Universal Robots PolyScope program: Hospital_small_top.urp

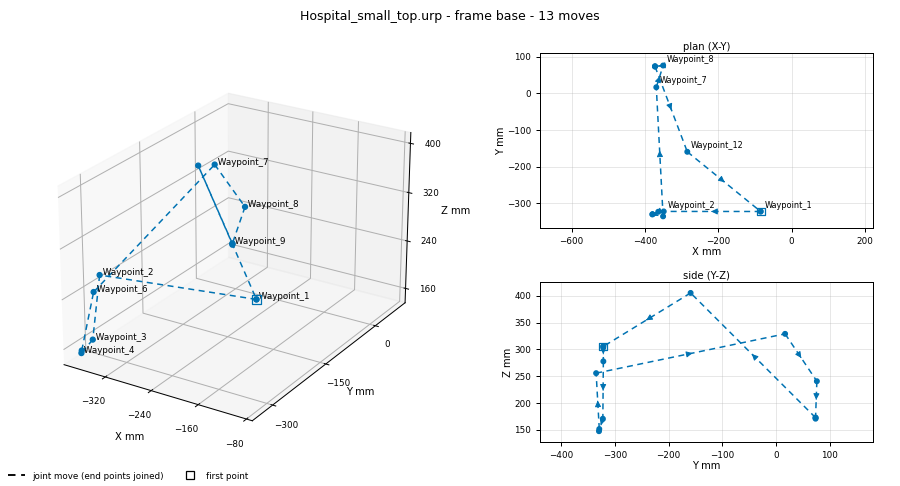
[picture p0: tool path of Hospital_small_top.urp in frame base, 13 of 13 moves have a stored position in this frame; points joined in program order, loops and branches not executed]
Program Hospital_small_top (installation=default directory=/programs/usbdisk/Zahra1 createdIn=5.11.11.1010533 lastSavedIn=5.11.11.1010533 robotSerialNumber=20205300864)
Calibrated DH parameters: a=[-0.000166, -0.243494, -0.153108, 0.000057, -0.000123, 0]; d=[0.151897, -1.34267, 53.988124, -52.514559, 0.085283, 0.092193]; alpha=[1.572472, -0.003756, 0.002824, 1.570807, -1.572621, 0]; deltaTheta=[0, 0.020704, 7.033215, -0.770746, 0.000004, 0]
Robot Program (runOnlyOnce=true)
  MoveJ speed 60 deg/s, acceleration 80 deg/s^2 (useActiveTCP=true) feature=Base
    Waypoint Waypoint_1: TCP in base x=-84.299 y=-321.882 z=305.489 mm, rx=-2.081 ry=-2.2572 rz=0.0985 rad; joints [-79.978, -91.2, -87.972, -91.694, 84.669, 815.507] deg
    URCap Gripper (Robotiq_Grippers, Robotiq Inc.) dataModel(position=41.96078431372549, force=70.0, speed=18.0, positionInDouble=41.96078431372549, forceInDouble=70.0, speedInDouble=18.0, slaveIds=[9], blocking=true, robotCompliant=false)
    Waypoint Waypoint_2: TCP in base x=-348.719 y=-321.719 z=277.773 mm, rx=-2.1945 ry=-2.1836 rz=0.1126 rad; joints [-120.615, -128.517, -45.514, -92.459, 86.402, 779.6] deg
    Waypoint Waypoint_3: TCP in base x=-363.621 y=-322.641 z=170.809 mm, rx=-2.1359 ry=-2.215 rz=0.1251 rad; joints [-121.994, -135.072, -63.231, -67.774, 85.458, 775.847] deg
    Waypoint Waypoint_4: TCP in base x=-379.661 y=-329.834 z=147.579 mm, rx=-2.2203 ry=-2.2148 rz=-0.0022 rad; joints [-123.935, -143.229, -52.439, -74.367, 89.583, 776.263] deg
    URCap Gripper (Robotiq_Grippers, Robotiq Inc.) dataModel(position=72.54901960784314, force=70.0, speed=18.0, positionInDouble=72.54901960784314, forceInDouble=70.0, speedInDouble=18.0, slaveIds=[9], blocking=true, robotCompliant=true)
    Waypoint Waypoint_5: motionParameters(jointSpeed=0.698132 jointAcceleration=0.349066 cartesianSpeed=0.25 cartesianAcceleration=1.2); TCP in base x=-379.309 y=-329.308 z=151.636 mm, rx=-2.2199 ry=-2.2154 rz=-0.0011 rad; joints [-123.934, -142.715, -52.326, -74.954, 89.584, 776.236] deg
    Waypoint Waypoint_6: TCP in base x=-350.417 y=-335.163 z=255.759 mm, rx=-2.1382 ry=-2.1875 rz=0.0356 rad; joints [-119.668, -133.183, -41.951, -94.671, 84.959, 779.051] deg
    Waypoint Waypoint_7: TCP in base x=-368.914 y=17.041 z=329.05 mm, rx=-3.1119 ry=-0.0989 rz=0.0771 rad; joints [-161.33, -100.25, -72.744, -94.639, 87.657, 825.065] deg
    Waypoint Waypoint_8: TCP in base x=-350.257 y=76.292 z=240.745 mm, rx=-3.1182 ry=-0.0304 rz=-0.021 rad; joints [-170.647, -100.353, -95.24, -75.268, 88.821, 818.378] deg
    Waypoint Waypoint_9: TCP in base x=-372.488 y=73.847 z=172.839 mm, rx=-3.1257 ry=0.0423 rz=-0.0774 rad; joints [-171.083, -112.188, -98.307, -62.338, 89.645, 820.641] deg
    Waypoint Waypoint_10: motionParameters(jointSpeed=0.698132 jointAcceleration=0.349066 cartesianSpeed=0.25 cartesianAcceleration=1.2); TCP in base x=-372.391 y=73.875 z=170.896 mm, rx=-3.1257 ry=0.0422 rz=-0.0774 rad; joints [-171.085, -112.404, -98.588, -61.841, 89.643, 820.635] deg
    URCap Gripper (Robotiq_Grippers, Robotiq Inc.) dataModel(position=56.86274509803921, force=50.0, speed=18.0, positionInDouble=56.86274509803921, forceInDouble=50.0, speedInDouble=18.0, slaveIds=[9], blocking=true, robotCompliant=false)
    URCap Gripper (Robotiq_Grippers, Robotiq Inc.) dataModel(position=31.764705882352942, force=50.0, speed=18.0, positionInDouble=31.764705882352942, forceInDouble=50.0, speedInDouble=18.0, slaveIds=[9], blocking=true, robotCompliant=true)
    Waypoint Waypoint_9: TCP in base x=-372.488 y=73.847 z=172.839 mm, rx=-3.1257 ry=0.0423 rz=-0.0774 rad; joints [-171.083, -112.188, -98.307, -62.338, 89.645, 820.641] deg
    Waypoint Waypoint_12: TCP in base x=-284.375 y=-159.038 z=405.306 mm, rx=3.0931 ry=0.4318 rz=-0.123 rad; joints [-126.324, -93.539, -59.586, -112.963, 87.359, 847.749] deg
    Waypoint Waypoint_1: TCP in base x=-84.299 y=-321.882 z=305.489 mm, rx=-2.081 ry=-2.2572 rz=0.0985 rad; joints [-79.978, -91.2, -87.972, -91.694, 84.669, 815.507] deg
